DATA_BLOCK "双向初始化_DB"
{ S7_Optimized_Access := 'TRUE' }
VERSION : 0.1
NON_RETAIN
"双向初始化"

BEGIN

END_DATA_BLOCK

